PROGRAM ASx
VAR
	PUMPMOTION: fbPumpMotion;
	WATCHDOG: fbWatchdogSwitching;
	RST: fbResetButton;
	CBL: fbFirealarm;
	AUT: fbFusealarm;
	JFB: fbJfb;
	OSP: fbOvervoltageProtection;
	GT3_NORR: fbOutDoorTempMean;
	MODBUS: fbModbusSekvensArray;
	SYSTEM: fbOaksSystem;
	(*
		Göteborg SP1 = 57.7089 SP2 = 11.9746 
		Stockholm SP1 = 59.3293 SP2 = 18.0686 
		Malmö SP1 = 55.6050 SP2 = 13.0038
		Karlstad SP1 = 59.4022 SP2 = 13.5115
		
		För att hitta andra städers koordinater googla "Vilka koordinater har STAD?"
	*)
	ASTRO: fbSunClock := (SP1 := 57.7089, SP2 := 11.9746); 
END_VAR
VAR_OUTPUT
	
END_VAR
VAR PERSISTENT

END_VAR

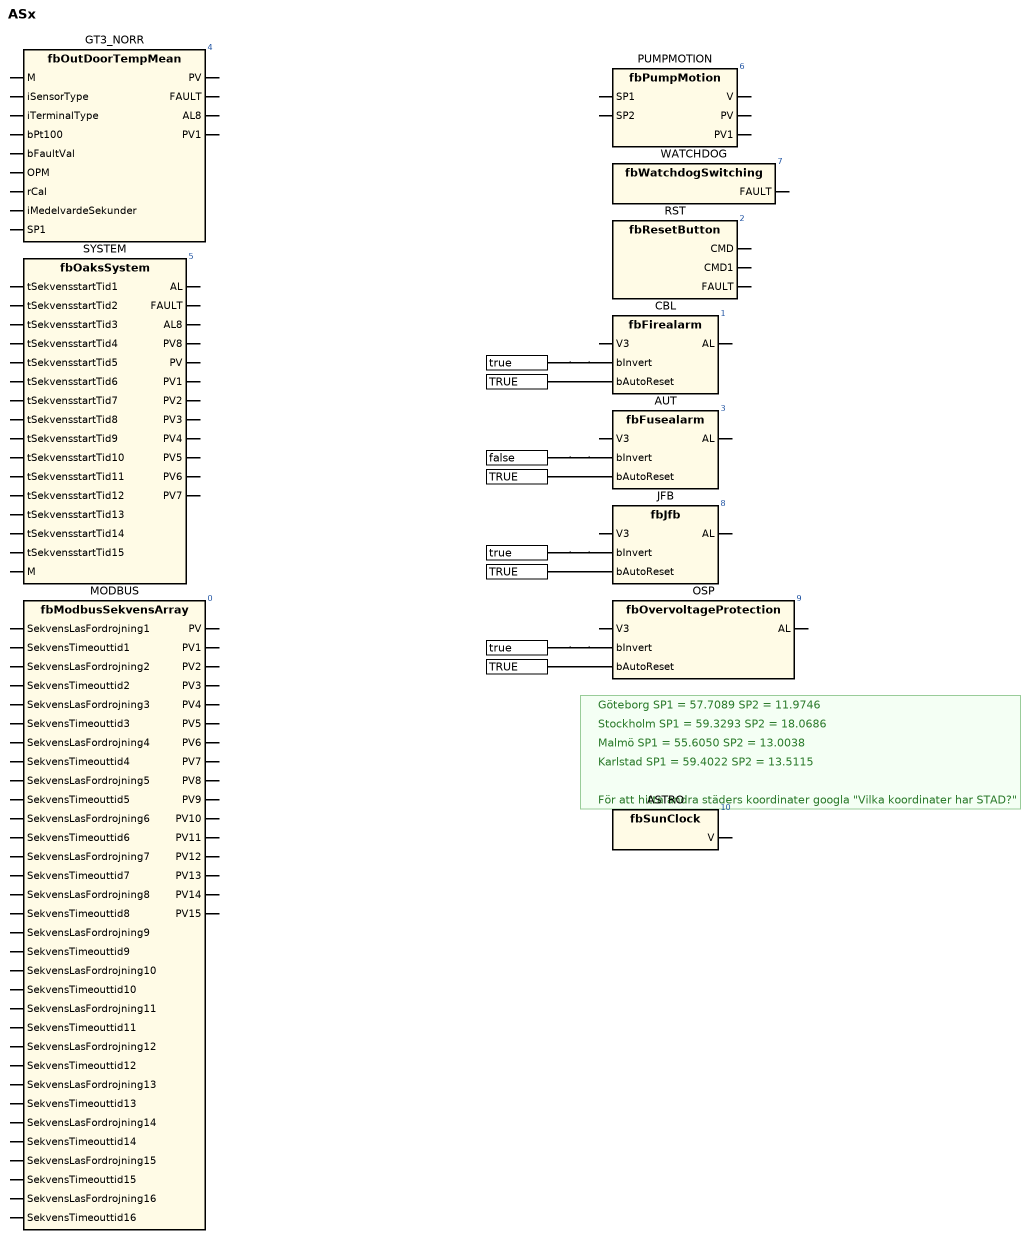
MODBUS(); // fbModbusSekvensArray
CBL(bInvert := true, bAutoReset := TRUE); // fbFirealarm
RST(); // fbResetButton
AUT(bInvert := false, bAutoReset := TRUE); // fbFusealarm
GT3_NORR(); // fbOutDoorTempMean
SYSTEM(); // fbOaksSystem
PUMPMOTION(); // fbPumpMotion
WATCHDOG(); // fbWatchdogSwitching
JFB(bInvert := true, bAutoReset := TRUE); // fbJfb
OSP(bInvert := true, bAutoReset := TRUE); // fbOvervoltageProtection
// 		Göteborg SP1 = 57.7089 SP2 = 11.9746
// 		Stockholm SP1 = 59.3293 SP2 = 18.0686
// 		Malmö SP1 = 55.6050 SP2 = 13.0038
// 		Karlstad SP1 = 59.4022 SP2 = 13.5115
//
// 		För att hitta andra städers koordinater googla "Vilka koordinater har STAD?"
ASTRO(); // fbSunClock

END_PROGRAM

(* stored: Version 1.1.0.1, ProductVersion 3.1.4022.18
   POU ASx: Id {27438f4d-ba85-41de-bb61-3ac6d62d36f6}, SpecialFunc None *)
